TYPE CM_Sensor_SIM :
STRUCT
END_STRUCT
END_TYPE

(* stored: Version 1.1.0.1, ProductVersion 3.1.4024.12
   DUT CM_Sensor_SIM: Id {cc3a7771-d953-438d-8db9-4c980008a031} *)
